FUNCTION SCODE_CODE : DWORD
VAR_INPUT
	sc		: DWORD;
END_VAR

SCODE_CODE := 16#FFFF AND sc;

END_FUNCTION

(* stored: Version 1.1.0.1, ProductVersion 3.1.4024.3
   POU SCODE_CODE: Id {986bae42-870a-484f-aa1f-b286e8d4d4c1}, SpecialFunc None *)
